TYPE "UDT_ZC_RECETA_CIP_RECHAZOS"
VERSION : 0.1
   STRUCT
      TiempoMaxDrenaje : Int := 0;   // RECHAZOS - Tiempo máximo de drenaje
      TiempoMaxEmpuje : Int := 0;   // RECHAZOS - Tiempo máximo de empuje
      ReservaInt_1 : Int;
      ConductividadDrenaje : Real := 0.0;   // RECHAZOS - Conductividad de drenaje
      ConductividadEmpuje : Real := 0.0;   // RECHAZOS - Conductividad de empuje
      ReservaReal_1 : Real;
   END_STRUCT;

END_TYPE

